TYPE ST_MethodArgumentData :
STRUCT
	eDataType		: E_UADataType;
	pData			: PVOID;
	nDataSize		: UINT;
	
END_STRUCT
END_TYPE

(* stored: Version 1.1.0.1, ProductVersion 3.1.4024.5
   DUT ST_MethodArgumentData: Id {6e870fbd-7d32-4ebc-8481-aae7c8c7fe38} *)
